{attribute 'qualified_only'}
VAR_GLOBAL CONSTANT
	MAX_BYTE_ARRAY : UINT := 255;
END_VAR

(* stored: Version 1.1.0.1, ProductVersion 3.1.4024.11
   GVL TcoVisionParams: Id {b1a1a2bf-e6ec-0090-3854-0486617c1e82}, ParameterList True *)
